FUNCTION_BLOCK E_CYCLE
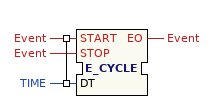
  EVENT_INPUT
    START WITH DT;
    STOP;
  END_EVENT
  EVENT_OUTPUT
    EO;
  END_EVENT
  VAR_INPUT
    DT : TIME;
  END_VAR
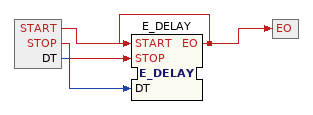
  FBS
    E_DELAY : E_DELAY;
  END_FBS
  EVENT_CONNECTIONS
    START TO E_DELAY.START;
    STOP TO E_DELAY.STOP;
    E_DELAY.EO TO E_DELAY.START;
    E_DELAY.EO TO EO;
  END_CONNECTIONS
  DATA_CONNECTIONS
    DT TO E_DELAY.DT;
  END_CONNECTIONS
END_FUNCTION_BLOCK
